Staubli VAL3: DecToBin.pgx

public program DecToBin(num x_nDecimal, string& x_sBinary[])
begin
  //-----------------------------------------------------------------------
  //Header begin
  //Description of program
  //  This program turns a decimal number into a binary word.
  //  Receives decimal value and turns it into the corresponding
  //  binary word.
  //
  //Input parameters
  //  num x_nDecimal :
  //    role : decimal value to convert
  //
  //Output parameters
  //  string x_sBinary :
  //    role : binary value converted
  //
  //Example
  //  DecToBin(42,sBinaryValue)
  //
  //History
  //  Creation : 16-04-09 - t.Gra
  //Header end
  //-----------------------------------------------------------------------
  //take the full value
  x_nDecimal=roundDown(x_nDecimal)
  //Calcul loop
  do
    if (x_nDecimal%2)==0
      x_sBinary="0"+x_sBinary
    else
      x_sBinary="1"+x_sBinary
    endIf
    x_nDecimal=roundDown(x_nDecimal/2)
  until (x_nDecimal<1)
end
